INTERFACE INTERNAL _I_Entity EXTENDS I_Debug, I_ValidateInterface

PROPERTY INTERNAL _Next : I_Entity
GET
END_GET
SET
END_SET
END_PROPERTY

PROPERTY INTERNAL _Prev : I_Entity
GET
END_GET
SET
END_SET
END_PROPERTY

PROPERTY INTERNAL _Raw : I_Generic
GET
END_GET
SET
END_SET
END_PROPERTY

PROPERTY INTERNAL _Result : Result
GET
END_GET
END_PROPERTY

PROPERTY INTERNAL _NewInstance : BOOL
GET
END_GET
SET
END_SET
END_PROPERTY

END_INTERFACE

(* stored: Version 1.1.0.1
   Itf _I_Entity: Id {1f3e5d12-6188-40e2-9c90-96da8b656fc4}
   Property _Next: Id {74a5b398-fcd6-40c3-938e-d42157f8245f}
   Get Get: Id {a2533393-55f2-4086-88be-812839c9a40a}
   Set Set: Id {1241208d-a4b6-407c-9e37-a8db489ebb16}
   Property _Prev: Id {0c22a104-d522-4990-8c49-426d346ef56d}
   Get Get: Id {25945637-4710-4ae5-8fee-582acdf2c107}
   Set Set: Id {80cf25da-628d-4f4d-b555-effaee3a9d58}
   Property _Raw: Id {ad7a9299-a825-4730-8ae0-d234bc888fae}
   Get Get: Id {0a6763bf-c621-4899-8a2d-9b2c4bd145a9}
   Set Set: Id {33898199-6d53-42c6-8e58-2c03b5d1cae0}
   Property _Result: Id {47d5d0aa-f4f4-4e2a-8520-91182f9d82fc}
   Get Get: Id {9c90b34f-7efb-4749-a987-26c1ad5633e1}
   Property _NewInstance: Id {8234272d-6167-4c34-9007-0e46cd80224e}
   Get Get: Id {3752a4de-625e-4260-ac74-1674fb725c12}
   Set Set: Id {97bb8f31-c579-4709-bd6f-7fa6af1be49f} *)
